FUNCTION Convert_BOOL_TO_DT : Hresult
VAR_INPUT
	in : BOOL;
	out : REFERENCE TO DT;
END_VAR
VAR
	converted : DT;
END_VAR

converted := BOOL_TO_DT(in);

IF (DT_TO_BOOL(converted) <> in) THEN
	Convert_BOOL_TO_DT := INCOMPATIBLE;
	RETURN;
END_IF

out := converted;

END_FUNCTION

(* stored: Version 1.1.0.1, ProductVersion 3.1.4024.12
   POU Convert_BOOL_TO_DT: Id {94abbb13-7185-4a03-b572-5b24ff5cd6db}, SpecialFunc None *)
